// TwinCAT 3 PLC project PLC1
// ProgramVersion: 3.1.4022.2
// libraries:
//   ERS_CO2 Payload Decoder, * (PXL-Tech)
//   MSC1608 Payload Decoder, * (PXL-Tech)
//   Tc2_EnOcean, * (Beckhoff Automation GmbH)
//   Tc2_Standard, * (Beckhoff Automation GmbH)
//   Tc2_System, * (Beckhoff Automation GmbH)
//   Tc2_TcpIp, * (Beckhoff Automation GmbH)
//   Tc2_Utilities, * (Beckhoff Automation GmbH)
//   Tc3_JsonXml, * (Beckhoff Automation GmbH)
//   Tc3_Module, * (Beckhoff Automation GmbH)
//   VisuSymbols,3.5.10.0,System
// project tree:
//   / GlobalTextList.TcGTLO, PlcTask.TcTTO (not stored), Visualization Manager.TcVMO (not stored), VISU_TASK.TcTTO
//   GVLs/ GVL1.TcGVL
//   POUs/ Beamer_Projectorscherm.TcPOU (not stored), MAIN.TcPOU, Aanwezigheids_lichten.TcPOU (not stored), SendCommands.TcPOU (not stored)
//   VISUs/ Visualization.TcVIS

CONFIGURATION PLC1
    RESOURCE PLC ON TwinCAT3
        TASK VISU_TASK(INTERVAL := T#200000us, PRIORITY := 30);
        PROGRAM VisuElems_Visu_Prg WITH VISU_TASK : VisuElems.Visu_Prg;
    END_RESOURCE
END_CONFIGURATION

// ---- GVLs/GVL1.TcGVL
VAR_GLOBAL
	
//lichtsturing
LichtenRAAMKANT AT %Q*: BOOL;
LichtenDEURKANT AT %Q*: BOOL;

AanwezigheidsdetectorRAAMKANT AT %I*: BOOL;
AanwezigheidsdetectorDEURKANT AT %I*: BOOL;

LichtsterkteDEUR AT %I*: INT;
LichtsterkteDEUR2 AT %I*: INT;
LichtsterkteBORD AT %I*: INT;
lichtsterkteBORD2 AT %I*: INT;
LINKERKNOP AT %I* : BOOL;
RECHTERKNOP AT %I* : BOOL;


//beamer & projectorschermsturing

BeamerAANKNOP AT %I* : BOOL;
BeamerUITKNOP AT %I* : BOOL;
Projectorscherm AT %Q* : BOOL;



socketconnectknop AT %I* : BOOL;
socketsendknop AT %I* : BOOL;



//raamsturing


stKL6581            : STR_KL6581;


//Lora
	sDatastring: STRING(500);
	
	Moteeui			: STRING;
	Appeui			: STRING;
	UserData		: ST_UserData;
	PayloadDecoded	: STRING;

	PayloadLength	: DINT;
	PayloadData		: ARRAY[1..100] OF BYTE;
	NullByte		: BYTE := 0;


END_VAR

// ---- POUs/MAIN.TcPOU
PROGRAM MAIN
VAR
END_VAR

Lichtsturing();
EnOcean();
Beamercontrol();
Tcp_ip();

END_PROGRAM

// ---- GlobalTextList.TcGTLO
TEXTLIST GlobalTextList
  820 = 'Bar : %d'
  42 = 'Beamer OFF'
  198 = 'Beamer ON'
  817 = 'Close'
  831 = 'Conection'
  492 = 'Connect'
  830 = 'Create'
  833 = 'Datum/Tijd : %s'
  787 = 'Deurkant'
  828 = 'Error'
  822 = 'Humidity : %d %'
  823 = 'Level x : %d'
  824 = 'Level y : %d'
  825 = 'Level z : %d'
  818 = 'Mesage ID : %d'
  816 = 'Payload : %s'
  774 = 'Raamkant'
  815 = 'Recieve'
  829 = 'Sensor ID : %s'
  819 = 'Status : %d'
  821 = 'Temp : %.2f °c'
  832 = 'Type sensor : '
  826 = 'VibAmp : %d'
  827 = 'VidFreq : %d'
END_TEXTLIST

// ---- VISUs/Visualization.TcVIS
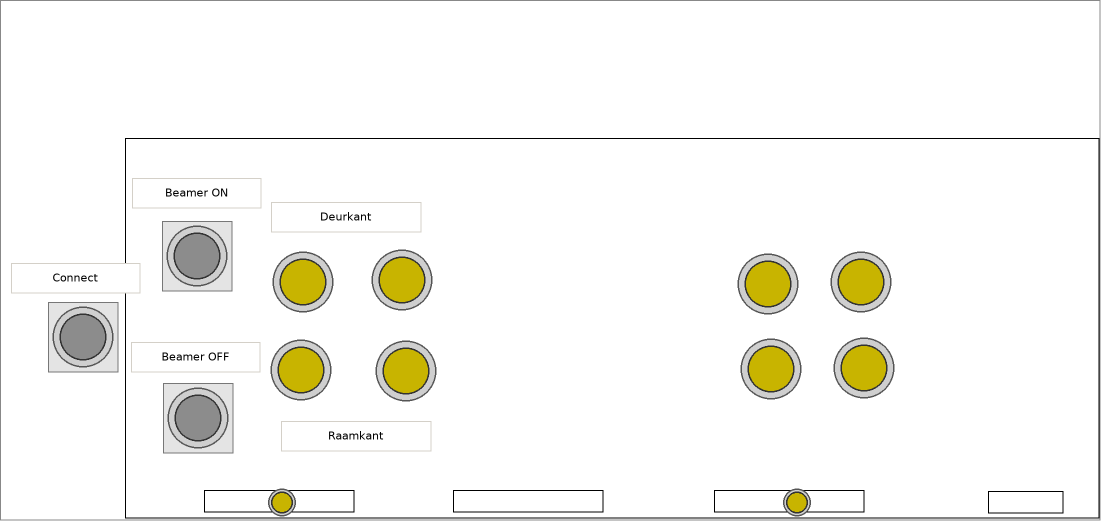
VISUALIZATION Visualization  // 1101x521
    Rectangle (125,138 974x380)
    Lamp1 (268,247 70x70), variable: Lichtsturing.relaisstandDEUR, style: Lamp-Lamp1-Yellow
    Lamp1 (367,245 70x70), variable: Lichtsturing.relaisstandDEUR, style: Lamp-Lamp1-Yellow
    Lamp1 (733,249 70x70), variable: Lichtsturing.relaisstandDEUR, style: Lamp-Lamp1-Yellow
    Lamp1 (826,247 70x70), variable: Lichtsturing.relaisstandDEUR, style: Lamp-Lamp1-Yellow
    Lamp1 (266,335 70x70), variable: Lichtsturing.relaisstandRAAM, style: Lamp-Lamp1-Yellow
    Lamp1 (371,336 70x70), variable: Lichtsturing.relaisstandRAAM, style: Lamp-Lamp1-Yellow
    Lamp1 (736,334 70x70), variable: Lichtsturing.relaisstandRAAM, style: Lamp-Lamp1-Yellow
    Lamp1 (829,333 70x70), variable: Lichtsturing.relaisstandRAAM, style: Lamp-Lamp1-Yellow
    Rectangle (204,490 150x22)
    Rectangle (453,490 150x22)
    Rectangle (714,490 150x22)
    Rectangle (988,491 75x22)
    Lamp1 (266,486 32x33), variable: EnOcean.raam2open, style: Lamp-Lamp1-Yellow
    Lamp1 (781,486 32x33), variable: EnOcean.raam1open, style: Lamp-Lamp1-Yellow
    Textfield (271,202 150x30), "Deurkant"
    Textfield (281,421 150x30), "Raamkant"
    PushSwitch (162,221 70x70), variable: BeamerAANKNOP, behaviour: TOGGLE, style: Switch-PushSwitch-Gray
    Textfield (132,178 129x30), "Beamer ON"
    PushSwitch (163,383 70x70), variable: BeamerUITKNOP, behaviour: TOGGLE, style: Switch-PushSwitch-Gray
    Textfield (131,342 129x30), "Beamer OFF"
    PushSwitch (48,302 70x70), variable: Beamercontrol.bconnect, behaviour: TOGGLE, style: Switch-PushSwitch-Gray
    Textfield (11,263 129x30), "Connect"
END_VISUALIZATION
